(* Single tank with LimitSwitchLow (piLsLow) and LimitSwitchHigh (piLsHigh)
| using this function when it have INDEPENDENT Measure weight
*)
FUNCTION_BLOCK FB_SingleTankSV1 EXTENDS FB_SingleTankS
VAR
	bAllowInMaterial : BOOL;
	bAllowOutMaterial : BOOL;
	lrLimitMinWeight : LREAL;
	lrLimitMaxWeight : LREAL;
	lrWeightWithdraw : LREAL; 		// weight withdraw Request
	lrWeightBeforeWD : LREAL;
	lrWeightWithdrawN : LREAL;
	lrWeight : LREAL;
	eState : E_TankState;
	iFill : I_TankFill;				// the components that action for fill materials.
	
	rTrigExecute : R_TRIG;
	bExecute : BOOL;//Execute with draw
	bFillError : BOOL;
	bError : BOOL;
	bWithDrawDone : BOOL;
	tonWithDrawStable : TON;
	tTimeWithDrawStable : TIME := T#3s; 
END_VAR

SUPER^();
rTrigExecute(CLK := bExecute);
bAllowOutMaterial := (lrWeight > lrLimitMinWeight);
bAllowInMaterial := (lrWeight < lrLimitMaxWeight);
lrWeightWithdrawN := lrWeightBeforeWD-lrWeight;
tonWithDrawStable(IN := eState=TANK_STOP, PT := tTimeWithDrawStable);
CASE eState OF
	TANK_IDLE:
		;// WAIT FOR CMD
	TANK_STOP:
		MS_Stop();
		
	TANK_WITHDRAWING:
		MS_Withdraw();
		
	TANK_FILLING:
		MS_Filling();
END_CASE

PROPERTY AllowIn : Reference to bool
GET
AllowIn ref= bAllowInMaterial;
END_GET
END_PROPERTY

(*
| Check the minimum condition  (lrWeight > lrLimitMinWeight
								AND piLslow.In;)
*)
PROPERTY AllowOut : REFERENCE TO BOOL
GET
AllowOut ref= bAllowOutMaterial;
END_GET
END_PROPERTY

METHOD AssignIfill : BOOL
VAR_INPUT
	iFill : I_TankFill;
END_VAR
THIS^.iFill := iFill;
END_METHOD

PROPERTY Error : reference to Bool
GET
Error ref= bError;
END_GET
END_PROPERTY

PROPERTY LimitMaxWeight : LREAL
GET
LimitMaxWeight := lrLimitMaxWeight;
END_GET
SET
lrLimitMaxWeight := LimitMaxWeight;
END_SET
END_PROPERTY

PROPERTY LimitMinWeight : LREAL
GET
LimitMinWeight := lrLimitMinWeight;
END_GET
SET
lrLimitMinWeight := LimitMinWeight;
END_SET
END_PROPERTY

METHOD MR_Filling : BOOL
VAR_INPUT
END_VAR
IF eState=TANK_IDLE 
	AND bAllowInMaterial
THEN
	eState := TANK_FILLING;
END_IF
END_METHOD

METHOD MR_Reset : BOOL
VAR_INPUT
END_VAR
bError := FALSE;
bWithDrawDone := FALSE;
MR_Reset := TRUE;
END_METHOD

METHOD MR_Stop : BOOL
VAR_INPUT
END_VAR
eState := TANK_STOP;
END_METHOD

(*	
	please call bExecute := false and then call bExecute := true for begin withdraw 
	if withdrawing => still withdraw
	else
		if not stop => MR_Stop before withdraw
*)
METHOD MR_WithDraw : BOOL
VAR_INPUT
	lrWeightWd : LREAL;
	bExecute : BOOL;
END_VAR
THIS^.bExecute := bExecute;
IF rTrigExecute.Q
	AND eState=TANK_IDLE 
	AND lrWeight > (lrWeightWd + lrLimitMinWeight) // Check enough weight
	AND bAllowOutMaterial
THEN
	eState := TANK_WITHDRAWING;
	lrWeightWithdraw := lrWeightWd;
	lrWeightBeforeWD := lrWeight;
END_IF
IF bExecute= FALSE THEN
	bWithDrawDone := FALSE;
END_IF
END_METHOD

METHOD PROTECTED MS_Filling
VAR_INPUT
END_VAR
IF bAllowInMaterial THEN
	iFill.Open();
ELSE
	iFill.Close();
	bError := TRUE;
	eState := TANK_STOP;
END_IF
END_METHOD

METHOD PROTECTED MS_Stop
VAR_INPUT
END_VAR
poCylinderCoil.Out := FALSE;
iFill.Close();
//bExecute := FALSE; // dont open this comment because it wrong.
IF tonWithDrawStable.Q THEN
	eState := TANK_IDLE;
END_IF
END_METHOD

METHOD PROTECTED MS_Withdraw
VAR_INPUT
END_VAR
poCylinderCoil.Out := TRUE;
IF lrWeightWithdrawN > lrWeightWithdraw THEN
	eState := TANK_STOP;
	bWithDrawDone := TRUE;
END_IF
IF NOT bAllowOutMaterial THEN
	bError := TRUE;
END_IF
END_METHOD

PROPERTY Ref_iFill : Reference to I_TankFill
GET
Ref_iFill ref= iFill;
END_GET
END_PROPERTY

PROPERTY TimeWithDrawStable : Time
GET
TimeWithDrawStable := tTimeWithDrawStable;
END_GET
SET
tTimeWithDrawStable := TimeWithDrawStable;
END_SET
END_PROPERTY

PROPERTY Weight : lreal
GET
Weight := lrWeight;
END_GET
SET
Weight := lrWeight;
END_SET
END_PROPERTY

PROPERTY WeightWithdraw : lreal
GET
WeightWithdraw := lrWeightWithdraw;
END_GET
SET
lrWeightWithdraw := WeightWithdraw;
END_SET
END_PROPERTY

PROPERTY WeightWithDrawN : lreal
GET
WeightWithDrawN := lrWeightWithdrawN;
END_GET
END_PROPERTY

PROPERTY WithDrawDone : Bool
GET
WithDrawDone := bWithDrawDone;
END_GET
END_PROPERTY

END_FUNCTION_BLOCK

(* stored: Version 1.1.0.1, ProductVersion 3.1.4024.12
   POU FB_SingleTankSV1: Id {5ca50686-0462-42c6-af5d-b0dee07be601}, SpecialFunc None
   Folder MR: Id {f1f24279-e1bb-479c-a8c0-d4ef91701c70}
   Folder MS: Id {4d7427c7-75e0-4a11-b8f5-045af82017e9}
   Property AllowIn: Id {19454c6c-9627-4b96-a378-44ef75eb1570}
   Get Get: Id {60617153-04c3-4fc2-9ae7-12ae57dedf08}
   Property AllowOut: Id {39f44b44-a9fa-435a-bb19-391cb7d16478}
   Get Get: Id {b20590ad-c50c-435a-9290-7ae3c5ce7d70}
   Method AssignIfill: Id {72d144b2-3662-4d8e-8e09-92841bd0d64b}
   Property Error: Id {7eb57e0c-d744-4ad7-b259-9cd03a95cd68}
   Get Get: Id {19a94231-4e98-4e6c-8bcf-4951ba35c618}
   Property LimitMaxWeight: Id {3d6dba06-1818-45ed-af6b-0451069573c3}
   Get Get: Id {b6cf597a-4d17-44f6-929d-51117270883c}
   Set Set: Id {da8fa2de-5e67-49c5-81d8-18fb7452fe09}
   Property LimitMinWeight: Id {b4e7bcc3-3741-428f-a558-a7ec417758e5}
   Get Get: Id {9222c5eb-6aac-4765-a7cd-79fa6d0e9eff}
   Set Set: Id {4bda1cf5-161a-4b71-8816-a4bdfad8340f}
   Method MR_Filling: Id {31dba4ab-4e68-42b2-8699-11e038c277bc}
   Method MR_Reset: Id {b7fbdb81-7ca2-40fb-8c0f-1c6b095064fc}
   Method MR_Stop: Id {8e0ae58f-f803-42bb-bfb2-c4909f9c3f1a}
   Method MR_WithDraw: Id {f46ebad8-bf4f-4fbd-bf93-7bd1b26757c7}
   Method MS_Filling: Id {bc9ac396-e513-4815-9e54-20b33958e075}
   Method MS_Stop: Id {7994ec05-7a9b-440c-8343-96d619b74c10}
   Method MS_Withdraw: Id {41ff54f8-9253-4da0-92c5-796eae7ab45c}
   Property Ref_iFill: Id {66f955d5-689a-4852-9b7e-e73d5da1c17f}
   Get Get: Id {425613c7-921f-4233-bfb0-0dc564f7c0db}
   Property TimeWithDrawStable: Id {fa79fd41-9f83-4c2c-9fec-2a2619a43c3e}
   Get Get: Id {73e5f184-89ca-4f11-9d90-56474f2014d4}
   Set Set: Id {119b3c97-119d-4472-922e-d187a18c7be6}
   Property Weight: Id {f9694997-df9d-4ef4-9fd1-d3c2a375fd1c}
   Get Get: Id {30b20208-6668-4802-acb5-9a350e95c5df}
   Set Set: Id {6f7db107-eab7-402a-9f99-ce491ba46a44}
   Property WeightWithdraw: Id {f9199ade-f15b-49a3-98e1-9236afd305a1}
   Get Get: Id {692b0709-82f1-4c92-80a5-618a2216c0cf}
   Set Set: Id {9acc50aa-9be8-440c-8df9-7dd6e10ff9fd}
   Property WeightWithDrawN: Id {705638db-f5aa-4651-8a66-8e4b22227b34}
   Get Get: Id {64a9aead-8c94-43a6-9a35-c2a6730978ea}
   Property WithDrawDone: Id {f8ac55f8-5350-4862-802b-c9681f46fd61}
   Get Get: Id {9b1551cd-8c19-4e9e-abd4-31415942af21} *)
